FUNCTION_BLOCK C_SERIALCOMM_PORT IMPLEMENTS I_SERIALCONTROLLER
VAR_INPUT
END_VAR
VAR_OUTPUT
END_VAR
VAR
	//Software Buffer
		_txbuffer 		: ComBuffer;
		_rxbuffer		: ComBuffer;	
	//Internal Memory Buffer
		_buffer 	: ARRAY[0..3000] OF BYTE;
	C_LINECONTROL 	: SerialLineControl;
	C_SendData 		: SendData;
	C_ReceiveData	: ReceiveData;
	_prefix, _suffix: STRING(15);
	_timeout 		: TIME := T#500MS;
END_VAR

METHOD UPDATE_BUFFER : DINT
{warning 'Hardware function is not implemented in Serial Comm base class'}
UPDATE_BUFFER := 0;
RETURN;
END_METHOD

PROPERTY RECEIVE_PREFIX : STRING(15)
SET
_prefix := prefix;
END_SET
GET
Prefix := _prefix;
END_GET
END_PROPERTY

METHOD SEND : DINT
VAR_INPUT
	ptr_data 	: PVOID;
	length		: UDINT;
END_VAR
C_SendData(
	pSendData:= ptr_data, 
	Length:= length, 
	TXbuffer:= _txbuffer);
IF C_SendData.Error <> COMERROR_NOERROR THEN
	Send := 1;
	RETURN;
ELSIF NOT C_SendData.Busy THEN
	Send := -1;
	RETURN;
ELSE
	Send := 0;
	RETURN;
END_IF
END_METHOD

METHOD RECEIVE : DINT
VAR_INPUT
	ptr_data 	: PVOID;
END_VAR
VAR
END_VAR
IF LEN(_prefix) > 0 THEN
	C_ReceiveData.pPrefix := ADR(_prefix);
	C_ReceiveData.LenPrefix := INT_TO_BYTE(LEN(_prefix));
ELSE
	C_ReceiveData.pPrefix := 0;
	C_ReceiveData.LenPrefix := 0;
END_IF
IF LEN(_suffix) > 0 THEN
	C_ReceiveData.pSuffix := ADR(_suffix);
	C_ReceiveData.LenSuffix := INT_TO_BYTE(LEN(_suffix));
ELSE
	C_ReceiveData.pSuffix := 0;
	C_ReceiveData.LenSuffix := 0;
END_IF
C_ReceiveData(
	pReceiveData:= ADR(_buffer), 
	SizeReceiveData:= SIZEOF(_buffer), 
	Timeout:= _timeout, 
	LenReceiveData=> , 
	RXbuffer:= _rxbuffer);
IF C_ReceiveData.Error <> COMERROR_NOERROR THEN
	Receive := 1;
	RETURN;
ELSIF C_ReceiveData.DataReceived THEN
	MEMCPY(ptr_data, ADR(_buffer), C_ReceiveData.LenReceiveData);
	Receive := -1;
	RETURN;
ELSE
	Receive := 0;
	RETURN;
END_IF
END_METHOD

PROPERTY TIMEOUT : TIME
GET
TimeOut := _timeout;
END_GET
SET
_timeout := timeout;
END_SET
END_PROPERTY

PROPERTY RECEIVE_SUFFIX : STRING(15)
GET
RECEIVE_SUFFIX := _suffix;
END_GET
SET
_suffix := RECEIVE_SUFFIX;
END_SET
END_PROPERTY

END_FUNCTION_BLOCK

(* stored: Version 1.1.0.1, ProductVersion 3.1.4020.3
   POU C_SERIALCOMM_PORT: Id {4e04354b-0238-4af2-9700-d58f6f2a81a4}, SpecialFunc None
   Folder Properties: Id {527a4af9-292e-4e17-b518-6a41f46b8a91}
   Folder Methods: Id {8f5898b1-49dd-4b6a-8a29-ef1dffc37d29}
   Method UPDATE_BUFFER: Id {36ad9a45-66b3-485f-9e4d-b0cad0792f89}
   Property RECEIVE_PREFIX: Id {384c528f-f7fc-4df3-a005-bb3804a0b3ee}
   Set Set: Id {37ec1fd1-2f33-4239-80f9-9b05ca3a5aa4}
   Get Get: Id {87cad6f4-9023-40d9-a671-1bfad9b8fc85}
   Method SEND: Id {3eb09680-9cfa-425f-b5f0-18dadaa85f69}
   Method RECEIVE: Id {810adef9-b34c-4f5a-9e46-6acf5bc716df}
   Property TIMEOUT: Id {bc87036c-275e-440d-8811-8ecad8d1b588}
   Get Get: Id {c0a741ee-d22f-4425-91b2-b00ac0e44f37}
   Set Set: Id {fd35c3f4-9282-4bd9-98b9-237a6e768049}
   Property RECEIVE_SUFFIX: Id {d004c93a-e11d-438c-9906-d3ef808796b8}
   Get Get: Id {2d6c18a7-6d66-416f-b01b-d6ec0a451a95}
   Set Set: Id {87c3cf67-019d-4a8e-85e4-db8e759b91c8} *)
